PROGRAM MAIN
VAR
END_VAR

END_PROGRAM

(* stored: Version 1.1.0.1
   POU MAIN: Id {247c4b0f-9579-4e4c-a952-4407e4dbe91c} *)
